PROGRAM PRG_MAIN
VAR
	
	fb_Antriebe : FB_Antriebe;
	fb_Betriebsart : FB_BA_Umschaltung;
	fbADSLogger		: FB_AdsLog;
	fbAmpel			: FB_Ampel;

END_VAR



fb_Betriebsart();
fb_Antriebe();
fbADSLogger();

fbAmpel(bBlinktakt := GVL_HMI_Ampel.bBlinktakt,
		btnReset:= GVL_HMI_Ampel.btnReset,
		btnActive := GVL_HMI_Ampel.btnActive,
		LED_ROT => GVL_HMI_Ampel.LED_Rot,
		LED_GELB => GVL_HMI_Ampel.LED_Gelb,
		LED_GRUEN => GVL_HMI_Ampel.LED_Gruen,
	config := GVL_Ampel.config[E_Ampeln.Lindesntrasse]);
		
GVL_A1.S01_C3_PF1 := fbAmpel.LED_ROT;
GVL_A1.S01_C3_PJ1 := fbAmpel.LED_ROT AND GVL_HMI_Ampel.bBlinktakt;
GVL_A1.S01_C3_PF2 := fbAmpel.LED_GELB;
GVL_A1.S01_C3_PF3 := fbAmpel.LED_GRUEN;

END_PROGRAM

(* stored: Version 1.1.0.1, ProductVersion 3.1.4024.12
   POU PRG_MAIN: Id {f327051d-30c9-411f-a87f-f29159a5f11e}, SpecialFunc None *)
